// TIA Portal V17 export
// export: Created 2025-03-07T09:16:31.6583242Z, ExportSetting WithDefaults, DisplayName Totally Integrated Automation Portal, DisplayVersion V17 Update 8, DisplayName TIA Portal Openness, DisplayVersion V17 Update 8, DisplayName TIA Portal Version Control Interface, DisplayVersion V17, DisplayName SINAMICS Startdrive Advanced, DisplayVersion V17 SP2, DisplayName SINAMICS Startdrive G110M, G120, G120C, G120D, G120P, G115D, DisplayVersion V17 SP2, DisplayName SINAMICS Startdrive G130, G150, S120, S150, SINAMICS MV, S210, DisplayVersion V17 SP2, DisplayName STEP 7 Professional, DisplayVersion V17 Update 8, DisplayName SINUMERIK ONE STEP 7 Toolbox, DisplayVersion V17 Update 12, DisplayName SINUMERIK 840D sl STEP 7 Toolbox, DisplayVersion V17 Update 12, DisplayName STEP 7 Safety, DisplayVersion V17 Update 6, DisplayName WinCC Advanced, DisplayVersion V17 Update 8
DATA_BLOCK "LBP_ModeGroup"   // DB11
TITLE = Mode group signals / Señales de grupo de modos de operación / Betriebsartengruppe Signale
{ S7_Optimized_Access := 'FALSE'; DB_Accessible_From_OPC_UA := 'FALSE' }
AUTHOR : SINUMERIK
FAMILY : SINUMERIK_ONE
VERSION : 6.15
// Interface between user program and mode groups, contains signals from/to the NC and operating software / Interfaz entre programa de usuario y grupos de modos de operación, contiene señales desde/hacia CN y software operativo. / Schnittstelle zwischen Anwenderprogramm und Betriebsartengruppen, enthält Signale von/zu NC and Betriebssoftware
// stored: AutoNumber false, DBAccessibleFromOPCUA false, DBAccessibleFromWebserver true, InstanceOfName LBP_typeModeGroup, InstanceOfType UDT, IsOnlyStoredInLoadMemory false, IsWriteProtectedInAS false
"LBP_typeModeGroup"
   // VAR RETAIN
   //    A_AUTO : Bool;
   //    A_MDA : Bool;
   //    A_JOG : Bool;
   //    f0_3 : Bool;
   //    A_MCDisable : Bool;
   //    A_MGStop : Bool;
   //    A_MGStopASp : Bool;
   //    A_MGReset : Bool;
   //    A_TEACHIN : Bool;
   //    A_REPOS : Bool;
   //    A_REF : Bool;
   //    f1_3 : Bool;
   //    f1_4 : Bool;
   //    f1_5 : Bool;
   //    A_SingleBlock_B : Bool;
   //    A_SingleBlock_A : Bool;
   //    A_INC1 : Bool;
   //    A_INC10 : Bool;
   //    A_INC100 : Bool;
   //    A_INC1000 : Bool;
   //    A_INC10000 : Bool;
   //    A_INCVar : Bool;
   //    A_ContManTravel : Bool;
   //    f2_7 : Bool;
   //    f3 : Byte;
   //    E_MMC_AUTO : Bool;
   //    E_MMC_MDA : Bool;
   //    E_MMC_JOG : Bool;
   //    f4_3 : Bool;
   //    f4_4 : Bool;
   //    f4_5 : Bool;
   //    f4_6 : Bool;
   //    f4_7 : Bool;
   //    E_MMC_TEACHIN : Bool;
   //    E_MMC_REPOS : Bool;
   //    E_MMC_REF : Bool;
   //    f5_3 : Bool;
   //    f5_4 : Bool;
   //    f5_5 : Bool;
   //    f5_6 : Bool;
   //    f5_7 : Bool;
   //    E_AUTO : Bool;
   //    E_MDA : Bool;
   //    E_JOG : Bool;
   //    E_MGOK : Bool;
   //    E_MGreseted : Bool;
   //    E_NCKintJOG : Bool;
   //    f6_6 : Bool;
   //    E_ChanReset : Bool;
   //    E_TEACHIN : Bool;
   //    E_REPOS : Bool;
   //    E_REF : Bool;
   //    f7_3 : Bool;
   //    f7_4 : Bool;
   //    f7_5 : Bool;
   //    f7_6 : Bool;
   //    f7_7 : Bool;
   //    E_INC1 : Bool;
   //    E_INC10 : Bool;
   //    E_INC100 : Bool;
   //    E_INC1000 : Bool;
   //    E_INC10000 : Bool;
   //    E_INCVar : Bool;
   //    E_ContManTravelAct : Bool;
   //    f8_7 : Bool;
   //    f9 : Byte;
   //    E_HMI_INC1 : Bool;
   //    E_HMI_INC10 : Bool;
   //    E_HMI_INC100 : Bool;
   //    E_HMI_INC1000 : Bool;
   //    E_HMI_INC10000 : Bool;
   //    E_HMI_INCVar : Bool;
   //    E_HMI_ContManTravel : Bool;
   //    f10_7 : Bool;
   //    f11 : Byte;
   //    f12 : Array[12..19] of Byte;
   //    MG : Array[2..10] of Struct
   //       A_AUTO : Bool;
   //       A_MDA : Bool;
   //       A_JOG : Bool;
   //       f0_3 : Bool;
   //       A_MCDisable : Bool;
   //       A_MGStop : Bool;
   //       A_MGStopASp : Bool;
   //       A_MGReset : Bool;
   //       A_TEACHIN : Bool;
   //       A_REPOS : Bool;
   //       A_REF : Bool;
   //       f1_3 : Bool;
   //       f1_4 : Bool;
   //       f1_5 : Bool;
   //       A_SingleBlock_B : Bool;
   //       A_SingleBlock_A : Bool;
   //       A_INC1 : Bool;
   //       A_INC10 : Bool;
   //       A_INC100 : Bool;
   //       A_INC1000 : Bool;
   //       A_INC10000 : Bool;
   //       A_INCVar : Bool;
   //       A_ContManTravel : Bool;
   //       f2_7 : Bool;
   //       f3 : Byte;
   //       E_MMC_AUTO : Bool;
   //       E_MMC_MDA : Bool;
   //       E_MMC_JOG : Bool;
   //       f4_3 : Bool;
   //       f4_4 : Bool;
   //       f4_5 : Bool;
   //       f4_6 : Bool;
   //       f4_7 : Bool;
   //       E_MMC_TEACHIN : Bool;
   //       E_MMC_REPOS : Bool;
   //       E_MMC_REF : Bool;
   //       f5_3 : Bool;
   //       f5_4 : Bool;
   //       f5_5 : Bool;
   //       f5_6 : Bool;
   //       f5_7 : Bool;
   //       E_AUTO : Bool;
   //       E_MDA : Bool;
   //       E_JOG : Bool;
   //       E_MGOK : Bool;
   //       E_MGreseted : Bool;
   //       E_NCKintJOG : Bool;
   //       f6_6 : Bool;
   //       E_ChanReset : Bool;
   //       E_TEACHIN : Bool;
   //       E_REPOS : Bool;
   //       E_REF : Bool;
   //       f7_3 : Bool;
   //       f7_4 : Bool;
   //       f7_5 : Bool;
   //       f7_6 : Bool;
   //       f7_7 : Bool;
   //       E_INC1 : Bool;
   //       E_INC10 : Bool;
   //       E_INC100 : Bool;
   //       E_INC1000 : Bool;
   //       E_INC10000 : Bool;
   //       E_INCVar : Bool;
   //       E_ContManTravelAct : Bool;
   //       f8_7 : Bool;
   //       f9 : Byte;
   //       E_HMI_INC1 : Bool;
   //       E_HMI_INC10 : Bool;
   //       E_HMI_INC100 : Bool;
   //       E_HMI_INC1000 : Bool;
   //       E_HMI_INC10000 : Bool;
   //       E_HMI_INCVar : Bool;
   //       E_HMI_ContManTravel : Bool;
   //       f10_7 : Bool;
   //       f11 : Byte;
   //       f12 : Array[12..19] of Byte;
   //    END_STRUCT;
   // END_VAR
BEGIN
END_DATA_BLOCK
